FUNCTION_BLOCK PUBLIC FB_SerialCommunication
VAR
	nInternalDatabits      : BYTE(7..8);
	eInternalParity        : E_Parity;
	nInternalStopbits	   : BYTE(1..2);	
END_VAR

;

{attribute 'monitoring' := 'call'}
PROPERTY PUBLIC Databits : BYTE(7..8)
GET
Databits := this^.nInternalDatabits;
END_GET
SET
this^.nInternalDatabits := Databits;
END_SET
END_PROPERTY

METHOD FB_init : BOOL
VAR_INPUT
	bInitRetains	: BOOL; // if TRUE, the retain variables are initialized (warm start / cold start)
	bInCopyCode		: BOOL; // if TRUE, the instance afterwards gets moved into the copy code (online change)
	nDatabits    	: BYTE(7..8);
	eParity         : E_Parity;
	nStopbits		: BYTE(1..2);
END_VAR
THIS^.nInternalDatabits := nDatabits;
THIS^.eInternalParity := eParity;
THIS^.nInternalStopbits := nStopbits;
END_METHOD

{attribute 'monitoring' := 'call'}
PROPERTY PUBLIC Parity : E_Parity
GET
Parity := THIS^.eInternalParity;
END_GET
SET
THIS^.eInternalParity := Parity;
END_SET
END_PROPERTY

{attribute 'monitoring' := 'call'}
PROPERTY PUBLIC Stopbits : BYTE(1..2)
GET
Stopbits := THIS^.nInternalStopbits;
END_GET
SET
THIS^.nInternalStopbits := Stopbits;
END_SET
END_PROPERTY

END_FUNCTION_BLOCK

(* stored: Version 1.1.0.1, ProductVersion 3.1.4022.18
   POU FB_SerialCommunication: Id {218335ff-386f-46ec-a884-7dee1a69d7c2}, SpecialFunc None
   Property Databits: Id {3ebbdef2-4871-4ed1-ba6e-01308a92d8e1}
   Get Get: Id {9f30611f-90db-4aca-b869-966e2918fe0f}
   Set Set: Id {1b40964b-b760-4af9-94c4-5130b09135fb}
   Method FB_init: Id {2e32824c-e8f6-491d-a5cf-e156585ea952}
   Property Parity: Id {ef01b680-49a0-4dff-a000-0a85a131c4ae}
   Get Get: Id {d9ebaa18-52c9-46ed-8e5c-44c18b14f7e7}
   Set Set: Id {c1dd8c42-ccba-44c6-9bff-360e67a5b463}
   Property Stopbits: Id {888ad274-0c71-442c-8b96-891fb56e56de}
   Get Get: Id {6c6e5b98-2053-4410-a83b-493154fbb6d0}
   Set Set: Id {7e1017cf-233f-41f5-a1fe-50ab64fc8785} *)
